// TIA Portal V16 export
// export: Created 2022-07-21T09:35:29.3408558Z, ExportSetting WithDefaults, DisplayName Totally Integrated Automation Portal, DisplayVersion V16 Update 4, DisplayName TIA Portal Version Control Interface, DisplayVersion V16 Update 2, DisplayName TIA Portal Openness, DisplayVersion V16 Update 4, DisplayName SINAMICS Startdrive Advanced, DisplayVersion V16 Update 5, DisplayName SINAMICS Startdrive G130, G150, S120, S150, SINAMICS MV, S210, DisplayVersion V16 Update 5, DisplayName SINAMICS Startdrive G110M, G120, G120C, G120D, G120P, G115D, DisplayVersion V16 Update 5, DisplayName STEP 7 Professional, DisplayVersion V16 Update 4, DisplayName STEP 7 Safety, DisplayVersion V16, DisplayName WinCC Advanced, DisplayVersion V16 Update 4
FUNCTION_BLOCK "fbInterrollLift"   // FB50, LAD
TITLE = Interroll lift handling / Obsługa windy Interroll
{ S7_Optimized_Access := 'TRUE' }
AUTHOR : a32thzz
VERSION : 0.1
// stored: AutoNumber true, IsIECCheckEnabled false, IsRetainMemResEnabled false, MemoryReserve 100, SetENOAutomatically false, UDAEnableTagReadback false
   VAR_INPUT
      disableAlarms : Bool;
      dataFromSafety : Bool;
      autoLiftUp : Bool;
      autoDriveRight : Bool;
      autoDriveLeft : Bool;
      hold : Bool := true;
      group : "typeGroup";
   END_VAR
   VAR_IN_OUT
      data : "typeInterrollUniversalFullLiftDrive";
   END_VAR
   VAR
      delayPTAlm0 : Time := T#5s;   // Czas opóźnienia dla alarmu 0 / delay alarm 0
      delayPTAlm1 : Time := T#1s;   // Czas opóźnienia dla alarmu 1 / delay alarm 1
      delayPTAlm2 : Time := T#1s;   // Czas opóźnienia dla alarmu 2 / delay alarm 2
      delayPTAlm3 : Time := T#1s;   // Czas opóźnienia dla alarmu 3 / delay alarm 3
      delayPTAlm4 : Time := T#1s;   // Czas opóźnienia dla alarmu 4 / delay alarm 4
      delayPTAlm5 : Time := T#1s;   // Czas opóźnienia dla alarmu 6 / delay alarm 6
      delayPTAlm6 : Time := T#1s;   // Czas opóźnienia dla alarmu 7 / delay alarm 7
      delayPTAlm7 : Time := T#1s;   // Czas opóźnienia dla alarmu 5 / delay alarm 5
      instTmrDlyAlm0 { S7_SetPoint := 'True'} : TON_TIME;   // Opóźnienie dla alarmu 0 / delay alarm 0
      instTmrDlyAlm1 { S7_SetPoint := 'True'} : TON_TIME;   // Opóźnienie dla alarmu 1 / delay alarm 1
      instTmrDlyAlm2 { S7_SetPoint := 'True'} : TON_TIME;   // Opóźnienie dla alarmu 2 / delay alarm 2
      instTmrDlyAlm3 { S7_SetPoint := 'True'} : TON_TIME;   // Opóźnienie dla alarmu 3 / delay alarm 3
      instTmrDlyAlm4 { S7_SetPoint := 'True'} : TON_TIME;   // Opóźnienie dla alarmu 4 / delay alarm 4
      instTmrDlyAlm5 { S7_SetPoint := 'True'} : TON_TIME;   // Opóźnienie dla alarmu 5 / delay alarm 5
      instTmrDlyAlm6 { S7_SetPoint := 'True'} : TON_TIME;   // Opóźnienie dla alarmu 7 / delay alarm 7
      instTmrDlyAlm7 { S7_SetPoint := 'True'} : TON_TIME;   // Opóźnienie dla alarmu 6 / delay alarm 6
      liftUpTON { S7_SetPoint := 'True'} : TON_TIME;   // Opóźnienie doajzdu do krańcówki / delay move to limit switch
   END_VAR
   VAR_TEMP
      bAlm0 : Bool;   // tymczasowy bit dla alarmu 0 / temporary alarm bit 0
      bAlm1 : Bool;   // tymczasowy bit dla alarmu 1 / temporary alarm bit 1
      bAlm2 : Bool;   // tymczasowy bit dla alarmu 2 / temporary alarm bit 2
      bAlm3 : Bool;   // tymczasowy bit dla alarmu 3 / temporary alarm bit 3
      bAlm4 : Bool;   // tymczasowy bit dla alarmu 4 / temporary alarm bit 4
      bAlm5 : Bool;   // tymczasowy bit dla alarmu 5 / temporary alarm bit 5
      bAlm6 : Bool;   // tymczasowy bit dla alarmu 6 / temporary alarm bit 6
      bAlm7 : Bool;   // tymczasowy bit dla alarmu 7 / temporary alarm bit 7
   END_VAR
BEGIN

REGION Network 1: Copy inputs -> structure / Przepisanie danych z wejść do struktury
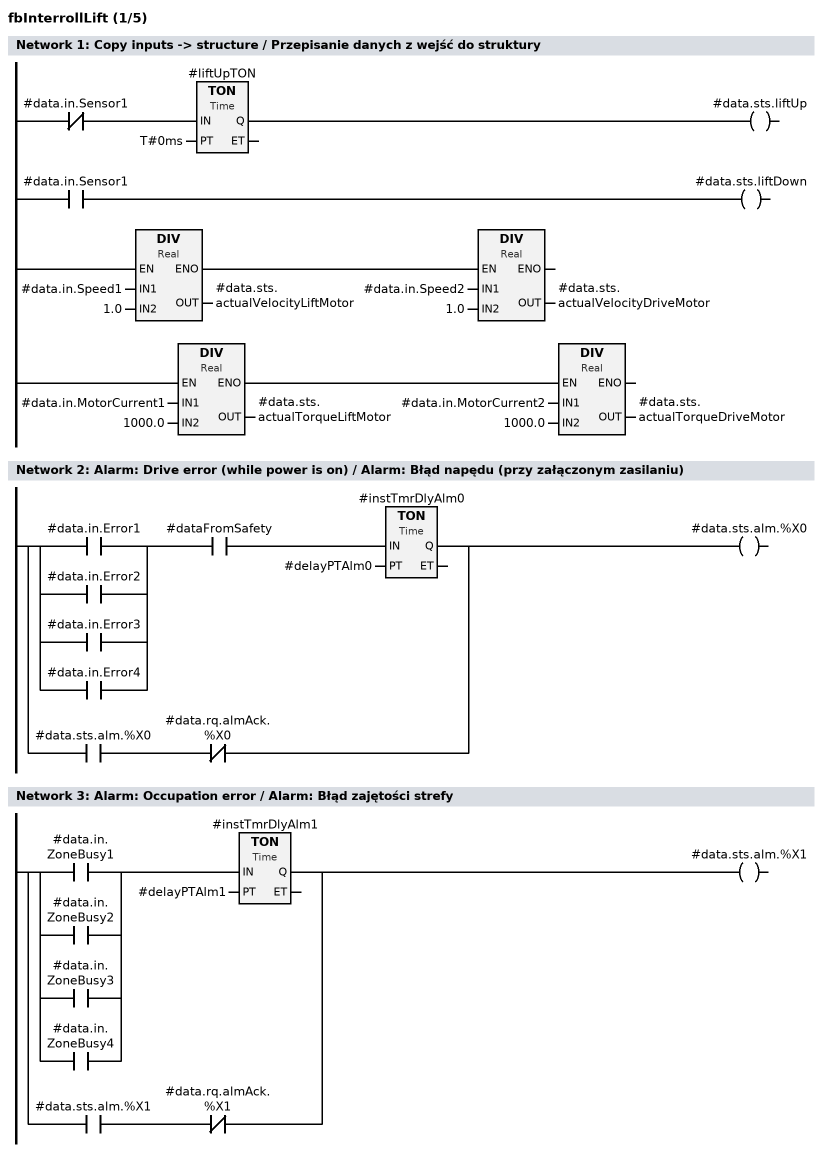
   RUNG wire#powerrail
      I_Contact( #data.in.Sensor1 )
      { S7_Templates := "time_type := Time" } #liftUpTON.TON(pt := T#0ms, et =>)
      Coil( #data.sts.liftUp )
   END_RUNG
   RUNG wire#powerrail
      Contact( #data.in.Sensor1 )
      Coil( #data.sts.liftDown )
   END_RUNG
   RUNG wire#powerrail
      { S7_Templates := "SrcType := Real" } Div(in1 := #data.in.Speed1, in2 := 1.0, out => #data.sts.actualVelocityLiftMotor)
      { S7_Templates := "SrcType := Real" } Div(in1 := #data.in.Speed2, in2 := 1.0, out => #data.sts.actualVelocityDriveMotor)
   END_RUNG
   RUNG wire#powerrail
      { S7_Templates := "SrcType := Real" } Div(in1 := #data.in.MotorCurrent1, in2 := 1000.0, out => #data.sts.actualTorqueLiftMotor)
      { S7_Templates := "SrcType := Real" } Div(in1 := #data.in.MotorCurrent2, in2 := 1000.0, out => #data.sts.actualTorqueDriveMotor)
   END_RUNG
   // the same network as SCL:
   #liftUpTON(IN := NOT #data.in.Sensor1, PT := T#0ms);   // TON
   #data.sts.liftUp := #liftUpTON.Q;
   #data.sts.liftDown := #data.in.Sensor1;
   #data.sts.actualVelocityLiftMotor := #data.in.Speed1 / 1.0;
   #data.sts.actualVelocityDriveMotor := #data.in.Speed2 / 1.0;
   #data.sts.actualTorqueLiftMotor := #data.in.MotorCurrent1 / 1000.0;
   #data.sts.actualTorqueDriveMotor := #data.in.MotorCurrent2 / 1000.0;
END_REGION

REGION Network 2: Alarm: Drive error (while power is on) / Alarm: Błąd napędu (przy załączonym zasilaniu)
   RUNG wire#powerrail
      Contact( #data.in.Error1 )
      wire#w1
      Contact( #dataFromSafety )
      { S7_Templates := "time_type := Time" } #instTmrDlyAlm0.TON(pt := #delayPTAlm0, et =>)
      wire#w2
      Coil( #data.sts.alm.%X0 )
   END_RUNG
   RUNG wire#powerrail
      Contact( #data.in.Error2 )
   END_RUNG wire#w1
   RUNG wire#powerrail
      Contact( #data.in.Error3 )
   END_RUNG wire#w1
   RUNG wire#powerrail
      Contact( #data.in.Error4 )
   END_RUNG wire#w1
   RUNG wire#powerrail
      Contact( #data.sts.alm.%X0 )
      I_Contact( #data.rq.almAck.%X0 )
   END_RUNG wire#w2
   // the same network as SCL:
   #instTmrDlyAlm0(IN := (#data.in.Error1 OR #data.in.Error2 OR #data.in.Error3 OR #data.in.Error4) AND #dataFromSafety,   // TON
                   PT := #delayPTAlm0);
   #data.sts.alm.%X0 := #instTmrDlyAlm0.Q OR (#data.sts.alm.%X0 AND NOT #data.rq.almAck.%X0);
END_REGION

REGION Network 3: Alarm: Occupation error / Alarm: Błąd zajętości strefy
   RUNG wire#powerrail
      Contact( #data.in.ZoneBusy1 )
      wire#w1
      { S7_Templates := "time_type := Time" } #instTmrDlyAlm1.TON(pt := #delayPTAlm1, et =>)
      wire#w2
      Coil( #data.sts.alm.%X1 )
   END_RUNG
   RUNG wire#powerrail
      Contact( #data.in.ZoneBusy2 )
   END_RUNG wire#w1
   RUNG wire#powerrail
      Contact( #data.in.ZoneBusy3 )
   END_RUNG wire#w1
   RUNG wire#powerrail
      Contact( #data.in.ZoneBusy4 )
   END_RUNG wire#w1
   RUNG wire#powerrail
      Contact( #data.sts.alm.%X1 )
      I_Contact( #data.rq.almAck.%X1 )
   END_RUNG wire#w2
   // the same network as SCL:
   #instTmrDlyAlm1(IN := #data.in.ZoneBusy1 OR #data.in.ZoneBusy2 OR #data.in.ZoneBusy3 OR #data.in.ZoneBusy4,   // TON
                   PT := #delayPTAlm1);
   #data.sts.alm.%X1 := #instTmrDlyAlm1.Q OR (#data.sts.alm.%X1 AND NOT #data.rq.almAck.%X1);
END_REGION

REGION Network 4: Alarm: Zone error / Alarm: Błąd strefy
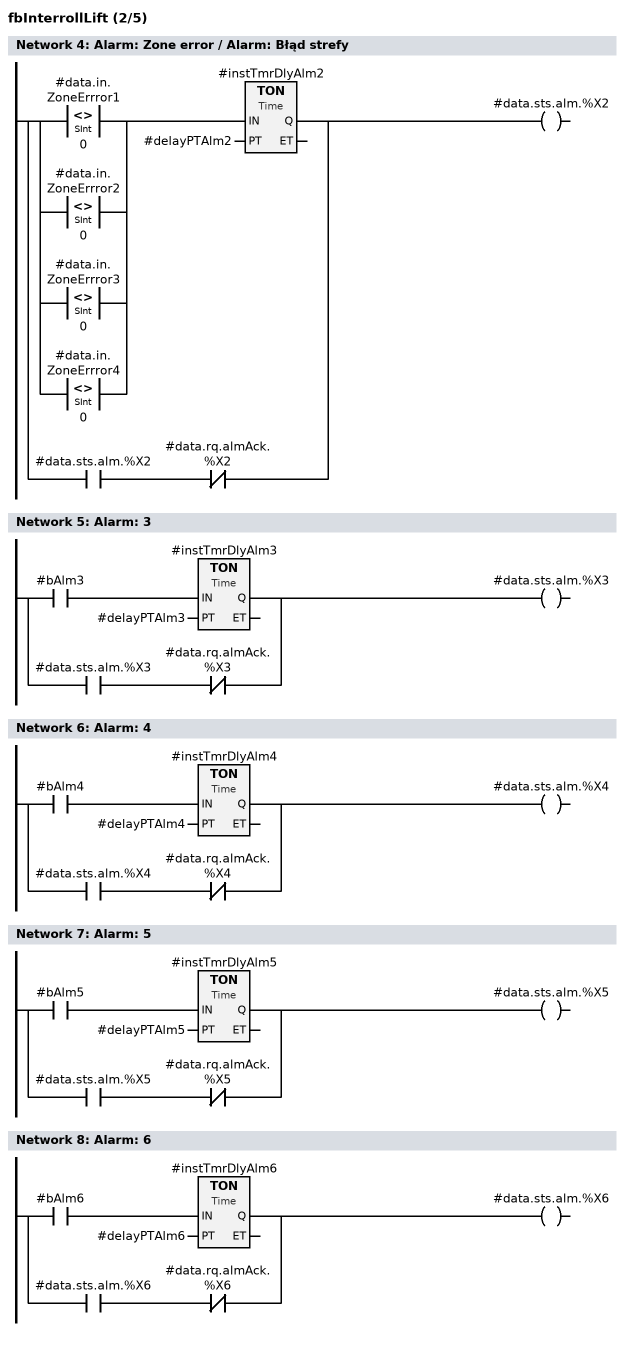
   RUNG wire#powerrail
      { S7_Templates := "SrcType := SInt" } NE_Contact(in1 := #data.in.ZoneErrror1, in2 := 0)
      wire#w1
      { S7_Templates := "time_type := Time" } #instTmrDlyAlm2.TON(pt := #delayPTAlm2, et =>)
      wire#w2
      Coil( #data.sts.alm.%X2 )
   END_RUNG
   RUNG wire#powerrail
      { S7_Templates := "SrcType := SInt" } NE_Contact(in1 := #data.in.ZoneErrror2, in2 := 0)
   END_RUNG wire#w1
   RUNG wire#powerrail
      { S7_Templates := "SrcType := SInt" } NE_Contact(in1 := #data.in.ZoneErrror3, in2 := 0)
   END_RUNG wire#w1
   RUNG wire#powerrail
      { S7_Templates := "SrcType := SInt" } NE_Contact(in1 := #data.in.ZoneErrror4, in2 := 0)
   END_RUNG wire#w1
   RUNG wire#powerrail
      Contact( #data.sts.alm.%X2 )
      I_Contact( #data.rq.almAck.%X2 )
   END_RUNG wire#w2
   // the same network as SCL:
   #instTmrDlyAlm2(IN := (#data.in.ZoneErrror1 <> 0) OR (#data.in.ZoneErrror2 <> 0) OR (#data.in.ZoneErrror3 <> 0) OR (#data.in.ZoneErrror4 <> 0),   // TON
                   PT := #delayPTAlm2);
   #data.sts.alm.%X2 := #instTmrDlyAlm2.Q OR (#data.sts.alm.%X2 AND NOT #data.rq.almAck.%X2);
END_REGION

REGION Network 5: Alarm: 3
   RUNG wire#powerrail
      Contact( #bAlm3 )
      { S7_Templates := "time_type := Time" } #instTmrDlyAlm3.TON(pt := #delayPTAlm3, et =>)
      wire#w1
      Coil( #data.sts.alm.%X3 )
   END_RUNG
   RUNG wire#powerrail
      Contact( #data.sts.alm.%X3 )
      I_Contact( #data.rq.almAck.%X3 )
   END_RUNG wire#w1
   // the same network as SCL:
   #instTmrDlyAlm3(IN := #bAlm3, PT := #delayPTAlm3);   // TON
   #data.sts.alm.%X3 := #instTmrDlyAlm3.Q OR (#data.sts.alm.%X3 AND NOT #data.rq.almAck.%X3);
END_REGION

REGION Network 6: Alarm: 4
   RUNG wire#powerrail
      Contact( #bAlm4 )
      { S7_Templates := "time_type := Time" } #instTmrDlyAlm4.TON(pt := #delayPTAlm4, et =>)
      wire#w1
      Coil( #data.sts.alm.%X4 )
   END_RUNG
   RUNG wire#powerrail
      Contact( #data.sts.alm.%X4 )
      I_Contact( #data.rq.almAck.%X4 )
   END_RUNG wire#w1
   // the same network as SCL:
   #instTmrDlyAlm4(IN := #bAlm4, PT := #delayPTAlm4);   // TON
   #data.sts.alm.%X4 := #instTmrDlyAlm4.Q OR (#data.sts.alm.%X4 AND NOT #data.rq.almAck.%X4);
END_REGION

REGION Network 7: Alarm: 5
   RUNG wire#powerrail
      Contact( #bAlm5 )
      { S7_Templates := "time_type := Time" } #instTmrDlyAlm5.TON(pt := #delayPTAlm5, et =>)
      wire#w1
      Coil( #data.sts.alm.%X5 )
   END_RUNG
   RUNG wire#powerrail
      Contact( #data.sts.alm.%X5 )
      I_Contact( #data.rq.almAck.%X5 )
   END_RUNG wire#w1
   // the same network as SCL:
   #instTmrDlyAlm5(IN := #bAlm5, PT := #delayPTAlm5);   // TON
   #data.sts.alm.%X5 := #instTmrDlyAlm5.Q OR (#data.sts.alm.%X5 AND NOT #data.rq.almAck.%X5);
END_REGION

REGION Network 8: Alarm: 6
   RUNG wire#powerrail
      Contact( #bAlm6 )
      { S7_Templates := "time_type := Time" } #instTmrDlyAlm6.TON(pt := #delayPTAlm6, et =>)
      wire#w1
      Coil( #data.sts.alm.%X6 )
   END_RUNG
   RUNG wire#powerrail
      Contact( #data.sts.alm.%X6 )
      I_Contact( #data.rq.almAck.%X6 )
   END_RUNG wire#w1
   // the same network as SCL:
   #instTmrDlyAlm6(IN := #bAlm6, PT := #delayPTAlm6);   // TON
   #data.sts.alm.%X6 := #instTmrDlyAlm6.Q OR (#data.sts.alm.%X6 AND NOT #data.rq.almAck.%X6);
END_REGION

REGION Network 9: Alarm: 7
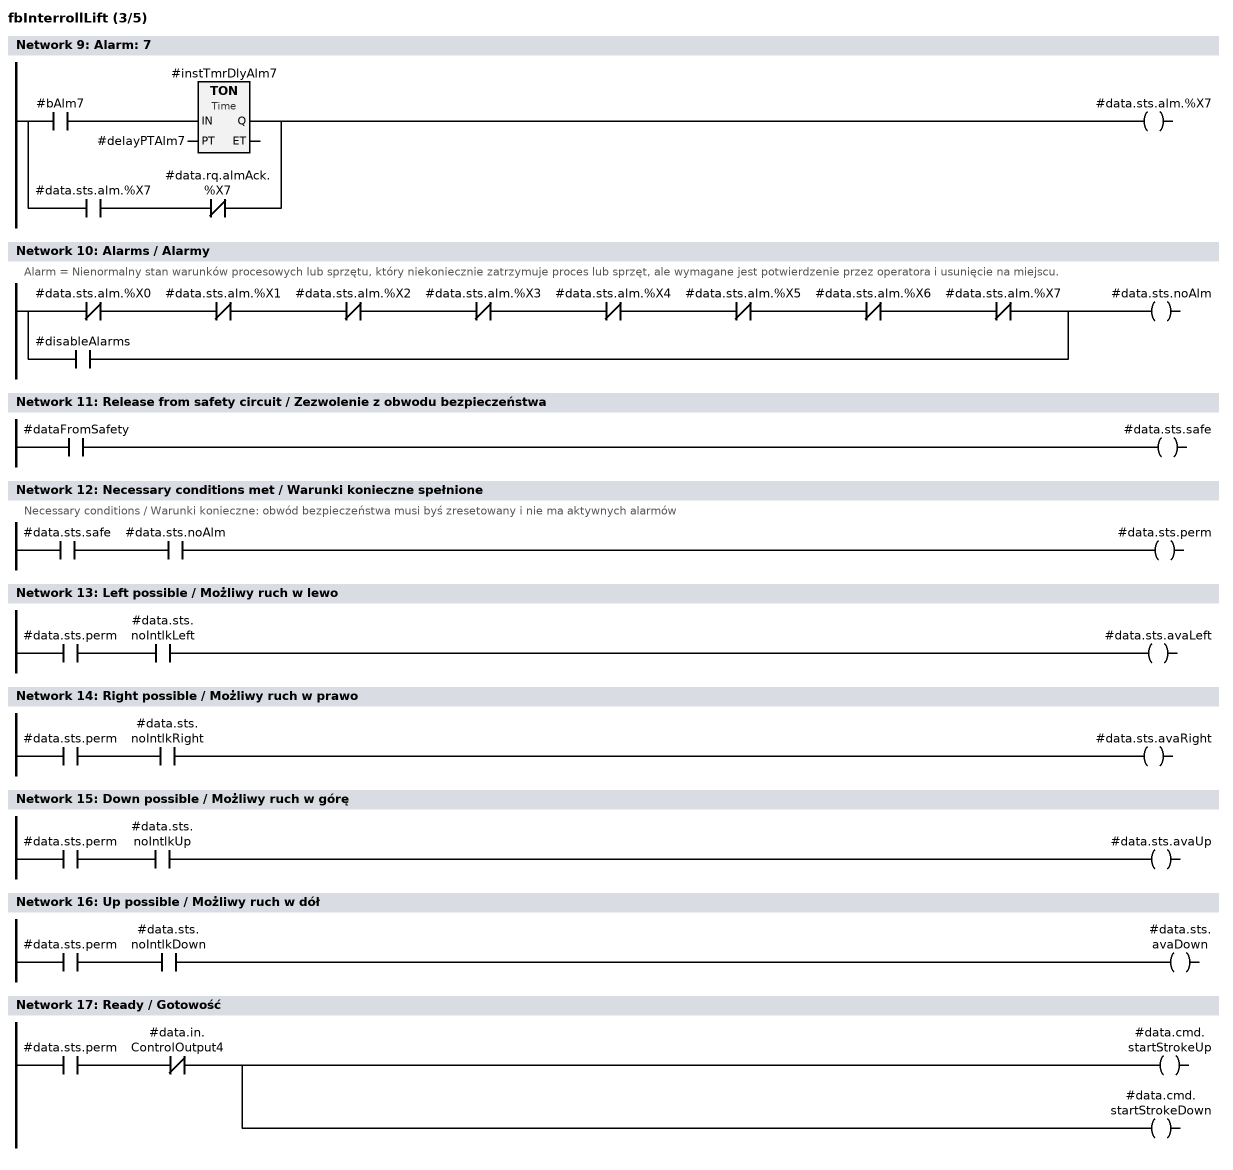
   RUNG wire#powerrail
      Contact( #bAlm7 )
      { S7_Templates := "time_type := Time" } #instTmrDlyAlm7.TON(pt := #delayPTAlm7, et =>)
      wire#w1
      Coil( #data.sts.alm.%X7 )
   END_RUNG
   RUNG wire#powerrail
      Contact( #data.sts.alm.%X7 )
      I_Contact( #data.rq.almAck.%X7 )
   END_RUNG wire#w1
   // the same network as SCL:
   #instTmrDlyAlm7(IN := #bAlm7, PT := #delayPTAlm7);   // TON
   #data.sts.alm.%X7 := #instTmrDlyAlm7.Q OR (#data.sts.alm.%X7 AND NOT #data.rq.almAck.%X7);
END_REGION

REGION Network 10: Alarms / Alarmy
   // Alarm = Nienormalny stan warunków procesowych lub sprzętu, który niekoniecznie zatrzymuje proces lub sprzęt, ale wymagane jest potwierdzenie przez operatora i usunięcie na miejscu.
   RUNG wire#powerrail
      I_Contact( #data.sts.alm.%X0 )
      I_Contact( #data.sts.alm.%X1 )
      I_Contact( #data.sts.alm.%X2 )
      I_Contact( #data.sts.alm.%X3 )
      I_Contact( #data.sts.alm.%X4 )
      I_Contact( #data.sts.alm.%X5 )
      I_Contact( #data.sts.alm.%X6 )
      I_Contact( #data.sts.alm.%X7 )
      wire#w1
      Coil( #data.sts.noAlm )
   END_RUNG
   RUNG wire#powerrail
      Contact( #disableAlarms )
   END_RUNG wire#w1
   // the same network as SCL:
   #data.sts.noAlm := (NOT #data.sts.alm.%X0 AND NOT #data.sts.alm.%X1 AND NOT #data.sts.alm.%X2 AND NOT #data.sts.alm.%X3 AND NOT #data.sts.alm.%X4 AND NOT #data.sts.alm.%X5 AND NOT #data.sts.alm.%X6 AND NOT #data.sts.alm.%X7) OR #disableAlarms;
END_REGION

REGION Network 11: Release from safety circuit / Zezwolenie z obwodu bezpieczeństwa
   RUNG wire#powerrail
      Contact( #dataFromSafety )
      Coil( #data.sts.safe )
   END_RUNG
   // the same network as SCL:
   #data.sts.safe := #dataFromSafety;
END_REGION

REGION Network 12: Necessary conditions met / Warunki konieczne spełnione
   // Necessary conditions / Warunki konieczne: obwód bezpieczeństwa musi byś zresetowany i nie ma aktywnych alarmów
   RUNG wire#powerrail
      Contact( #data.sts.safe )
      Contact( #data.sts.noAlm )
      Coil( #data.sts.perm )
   END_RUNG
   // the same network as SCL:
   #data.sts.perm := #data.sts.safe AND #data.sts.noAlm;
END_REGION

REGION Network 13: Left possible / Możliwy ruch w lewo
   RUNG wire#powerrail
      Contact( #data.sts.perm )
      Contact( #data.sts.noIntlkLeft )
      Coil( #data.sts.avaLeft )
   END_RUNG
   // the same network as SCL:
   #data.sts.avaLeft := #data.sts.perm AND #data.sts.noIntlkLeft;
END_REGION

REGION Network 14: Right possible / Możliwy ruch w prawo
   RUNG wire#powerrail
      Contact( #data.sts.perm )
      Contact( #data.sts.noIntlkRight )
      Coil( #data.sts.avaRight )
   END_RUNG
   // the same network as SCL:
   #data.sts.avaRight := #data.sts.perm AND #data.sts.noIntlkRight;
END_REGION

REGION Network 15: Down possible / Możliwy ruch w górę
   RUNG wire#powerrail
      Contact( #data.sts.perm )
      Contact( #data.sts.noIntlkUp )
      Coil( #data.sts.avaUp )
   END_RUNG
   // the same network as SCL:
   #data.sts.avaUp := #data.sts.perm AND #data.sts.noIntlkUp;
END_REGION

REGION Network 16: Up possible / Możliwy ruch w dół
   RUNG wire#powerrail
      Contact( #data.sts.perm )
      Contact( #data.sts.noIntlkDown )
      Coil( #data.sts.avaDown )
   END_RUNG
   // the same network as SCL:
   #data.sts.avaDown := #data.sts.perm AND #data.sts.noIntlkDown;
END_REGION

REGION Network 17: Ready / Gotowość
   RUNG wire#powerrail
      Contact( #data.sts.perm )
      I_Contact( #data.in.ControlOutput4 )
      wire#w1
      Coil( #data.cmd.startStrokeUp )
   END_RUNG
   RUNG wire#w1
      Coil( #data.cmd.startStrokeDown )
   END_RUNG
   // the same network as SCL:
   #data.cmd.startStrokeUp := #data.sts.perm AND NOT #data.in.ControlOutput4;
   #data.cmd.startStrokeDown := #data.cmd.startStrokeUp;
END_REGION

REGION Network 18: Move up / Ruch w górę
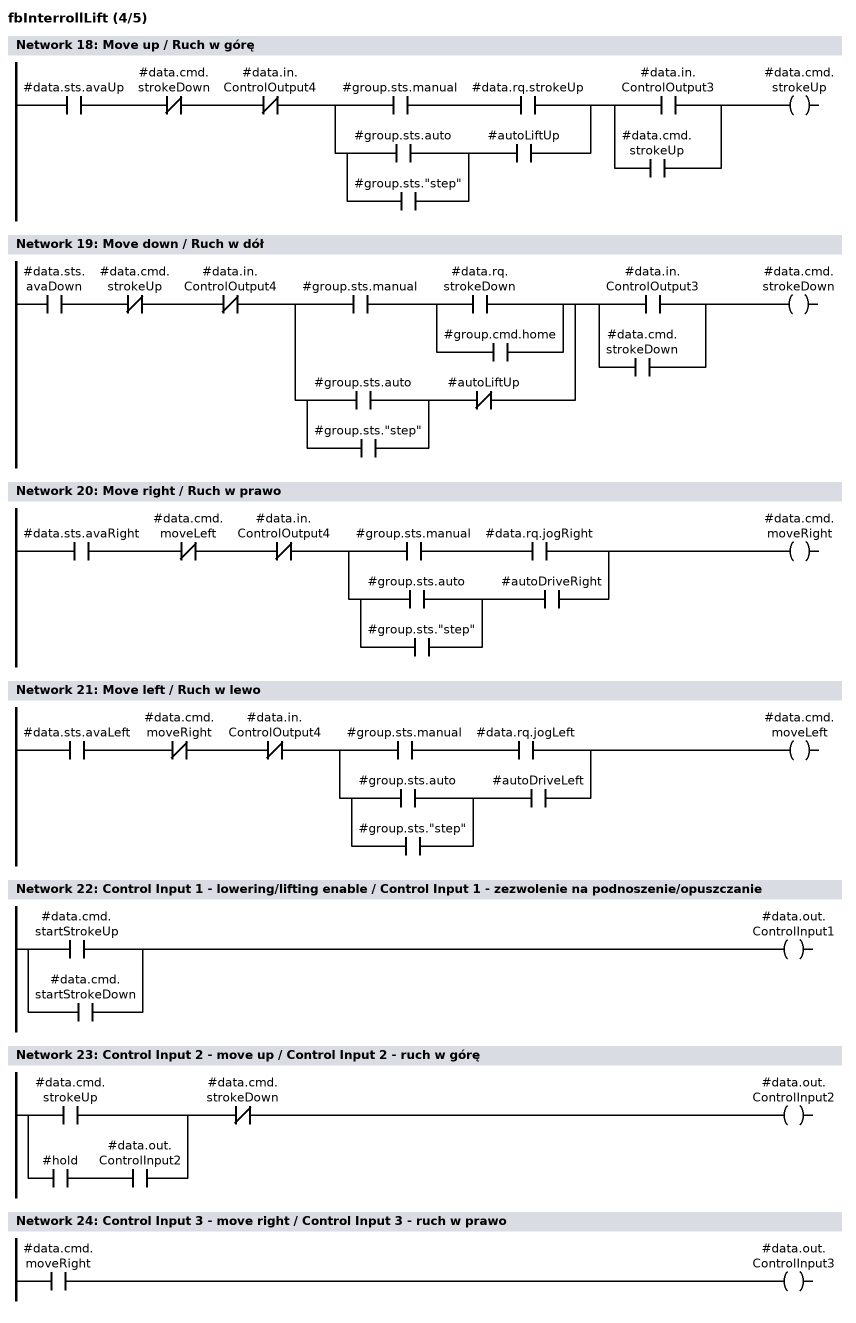
   RUNG wire#powerrail
      Contact( #data.sts.avaUp )
      I_Contact( #data.cmd.strokeDown )
      I_Contact( #data.in.ControlOutput4 )
      wire#w1
      Contact( #group.sts.manual )
      Contact( #data.rq.strokeUp )
      wire#w2
      Contact( #data.in.ControlOutput3 )
      wire#w4
      Coil( #data.cmd.strokeUp )
   END_RUNG
   RUNG wire#w1
      Contact( #group.sts.auto )
      wire#w3
      Contact( #autoLiftUp )
   END_RUNG wire#w2
   RUNG wire#w1
      Contact( #group.sts."step" )
   END_RUNG wire#w3
   RUNG wire#w2
      Contact( #data.cmd.strokeUp )
   END_RUNG wire#w4
   // the same network as SCL:
   #data.cmd.strokeUp := #data.sts.avaUp AND NOT #data.cmd.strokeDown AND NOT #data.in.ControlOutput4 AND ((#group.sts.manual AND #data.rq.strokeUp) OR ((#group.sts.auto OR #group.sts."step") AND #autoLiftUp)) AND (#data.in.ControlOutput3 OR #data.cmd.strokeUp);
END_REGION

REGION Network 19: Move down / Ruch w dół
   RUNG wire#powerrail
      Contact( #data.sts.avaDown )
      I_Contact( #data.cmd.strokeUp )
      I_Contact( #data.in.ControlOutput4 )
      wire#w1
      Contact( #group.sts.manual )
      wire#w2
      Contact( #data.rq.strokeDown )
      wire#w3
      Contact( #data.in.ControlOutput3 )
      wire#w5
      Coil( #data.cmd.strokeDown )
   END_RUNG
   RUNG wire#w2
      Contact( #group.cmd.home )
   END_RUNG wire#w3
   RUNG wire#w1
      Contact( #group.sts.auto )
      wire#w4
      I_Contact( #autoLiftUp )
   END_RUNG wire#w3
   RUNG wire#w1
      Contact( #group.sts."step" )
   END_RUNG wire#w4
   RUNG wire#w3
      Contact( #data.cmd.strokeDown )
   END_RUNG wire#w5
   // the same network as SCL:
   #data.cmd.strokeDown := #data.sts.avaDown AND NOT #data.cmd.strokeUp AND NOT #data.in.ControlOutput4 AND ((#group.sts.manual AND (#data.rq.strokeDown OR #group.cmd.home)) OR ((#group.sts.auto OR #group.sts."step") AND NOT #autoLiftUp)) AND (#data.in.ControlOutput3 OR #data.cmd.strokeDown);
END_REGION

REGION Network 20: Move right / Ruch w prawo
   RUNG wire#powerrail
      Contact( #data.sts.avaRight )
      I_Contact( #data.cmd.moveLeft )
      I_Contact( #data.in.ControlOutput4 )
      wire#w1
      Contact( #group.sts.manual )
      Contact( #data.rq.jogRight )
      wire#w2
      Coil( #data.cmd.moveRight )
   END_RUNG
   RUNG wire#w1
      Contact( #group.sts.auto )
      wire#w3
      Contact( #autoDriveRight )
   END_RUNG wire#w2
   RUNG wire#w1
      Contact( #group.sts."step" )
   END_RUNG wire#w3
   // the same network as SCL:
   #data.cmd.moveRight := #data.sts.avaRight AND NOT #data.cmd.moveLeft AND NOT #data.in.ControlOutput4 AND ((#group.sts.manual AND #data.rq.jogRight) OR ((#group.sts.auto OR #group.sts."step") AND #autoDriveRight));
END_REGION

REGION Network 21: Move left / Ruch w lewo
   RUNG wire#powerrail
      Contact( #data.sts.avaLeft )
      I_Contact( #data.cmd.moveRight )
      I_Contact( #data.in.ControlOutput4 )
      wire#w1
      Contact( #group.sts.manual )
      Contact( #data.rq.jogLeft )
      wire#w2
      Coil( #data.cmd.moveLeft )
   END_RUNG
   RUNG wire#w1
      Contact( #group.sts.auto )
      wire#w3
      Contact( #autoDriveLeft )
   END_RUNG wire#w2
   RUNG wire#w1
      Contact( #group.sts."step" )
   END_RUNG wire#w3
   // the same network as SCL:
   #data.cmd.moveLeft := #data.sts.avaLeft AND NOT #data.cmd.moveRight AND NOT #data.in.ControlOutput4 AND ((#group.sts.manual AND #data.rq.jogLeft) OR ((#group.sts.auto OR #group.sts."step") AND #autoDriveLeft));
END_REGION

REGION Network 22: Control Input 1 - lowering/lifting enable / Control Input 1 - zezwolenie na podnoszenie/opuszczanie
   RUNG wire#powerrail
      Contact( #data.cmd.startStrokeUp )
      wire#w1
      Coil( #data.out.ControlInput1 )
   END_RUNG
   RUNG wire#powerrail
      Contact( #data.cmd.startStrokeDown )
   END_RUNG wire#w1
   // the same network as SCL:
   #data.out.ControlInput1 := #data.cmd.startStrokeUp OR #data.cmd.startStrokeDown;
END_REGION

REGION Network 23: Control Input 2 - move up / Control Input 2 - ruch w górę
   RUNG wire#powerrail
      Contact( #data.cmd.strokeUp )
      wire#w1
      I_Contact( #data.cmd.strokeDown )
      Coil( #data.out.ControlInput2 )
   END_RUNG
   RUNG wire#powerrail
      Contact( #hold )
      Contact( #data.out.ControlInput2 )
   END_RUNG wire#w1
   // the same network as SCL:
   #data.out.ControlInput2 := (#data.cmd.strokeUp OR (#hold AND #data.out.ControlInput2)) AND NOT #data.cmd.strokeDown;
END_REGION

REGION Network 24: Control Input 3 - move right / Control Input 3 - ruch w prawo
   RUNG wire#powerrail
      Contact( #data.cmd.moveRight )
      Coil( #data.out.ControlInput3 )
   END_RUNG
   // the same network as SCL:
   #data.out.ControlInput3 := #data.cmd.moveRight;
END_REGION

REGION Network 25: Control Input 4 - move left / Control Input 4 - ruch w lewo
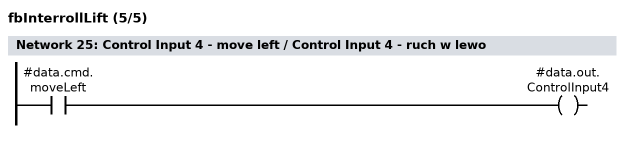
   RUNG wire#powerrail
      Contact( #data.cmd.moveLeft )
      Coil( #data.out.ControlInput4 )
   END_RUNG
   // the same network as SCL:
   #data.out.ControlInput4 := #data.cmd.moveLeft;
END_REGION
END_FUNCTION_BLOCK
